// TIA Portal V19 export
VAR_GLOBAL   // PLC tag table "MODULE_SIZE"
   pointNull AT %MD8000 : DWord;
   setNull AT %MD8004 : DWord;
END_VAR
VAR_GLOBAL CONSTANT   // user constants
   M_AIN : Int := 0;
   M_ADIN : Int := 0;
   M_CVLV : Int := 0;
   M_DIFF : Int := 0;
   M_DIN : Int := 0;
   M_MTR : Int := 0;
   M_MTRDIR : Int := 0;
   M_MTRLIN : Int := 0;
   M_VLV : Int := 0;
   MAX_ADIN : Int := 23;
   MAX_AIN : Int := 199;
   MAX_DIFF : Int := 31;
   MAX_DIN : Int := 23;
   MAX_MTR : Int := 199;
   MAX_MTRDIR : Int := 199;
   MAX_MTRLIN : Int := 79;
   MAX_VLV : Int := 199;
   MAX_CVLV : Int := 31;
   MAX_PLANT : Int := 23;
   M_PLANT : Int := 1;
END_VAR
